{attribute 'GeneratedUsingTerminal: EL7201-0001-0017'}
{attribute addProperty BoxType "EL7201-0001-0017"}
{attribute addProperty Id "DS402_StatuswordAT %I*DS402_Statusword_9B36FDFC2DS402_Position_actual_valueAT %I*DS402_Position_actual_value_07DC4C744DS402_ControlwordAT %Q*DS402_Controlword_F3F147212DS402_Target_velocityAT %Q*DS402_Target_velocity_08A9583B4WcStateAT %I*WcState_9091E0EB2InfoDataAT %I*InfoData_DEBFC8B711"}
{attribute addProperty CRC "608787240"}
{attribute addProperty Size "25"}
TYPE EL7201_24495B28 EXTENDS EtcSlaveTerminalBase_947E5A46 :
STRUCT
	{attribute addProperty Name "DS402_Statusword"}
	DS402_Statusword : DS402_Statusword_9B36FDFC;
	{attribute addProperty Name "DS402_Position_actual_value"}
	DS402_Position_actual_value : DS402_Position_actual_value_07DC4C74;
	{attribute addProperty Name "DS402_Controlword"}
	DS402_Controlword : DS402_Controlword_F3F14721;
	{attribute addProperty Name "DS402_Target_velocity"}
	DS402_Target_velocity : DS402_Target_velocity_08A9583B;
	{attribute addProperty Name "WcState"}
	WcState : WcState_9091E0EB;
	{attribute addProperty Name "InfoData"}
	InfoData : InfoData_DEBFC8B7;
END_STRUCT
END_TYPE

(* stored: Version 1.2.0.0, ProductVersion 3.1.4024.9
   DUT EL7201_24495B28: Id {24d6f6c1-162d-4d44-b798-817de0baf137} *)
